// TIA Portal V17 export
// export: Created 2022-12-09T10:51:17.8914312Z, ExportSetting WithDefaults, DisplayName Totally Integrated Automation Portal, DisplayVersion V17 Update 5, DisplayName TIA Portal Openness, DisplayVersion V17 Update 5, DisplayName TIA Portal Version Control Interface, DisplayVersion V17, DisplayName Simotion SCOUT TIA, DisplayVersion 5.4.3.0, DisplayName SINAMICS Startdrive Advanced, DisplayVersion V17 SP1, DisplayName SINAMICS Startdrive G130, G150, S120, S150, SINAMICS MV, S210, DisplayVersion V17 SP1, DisplayName SINAMICS Startdrive G110M, G120, G120C, G120D, G120P, G115D, DisplayVersion V17 SP1, DisplayName STEP 7 Professional, DisplayVersion V17 Update 5, DisplayName STEP 7 Safety, DisplayVersion V17, DisplayName WinCC Advanced, DisplayVersion V17 Update 5
TYPE "UDT_OMAC_GlobalData"
// stored: IsFailsafeCompliant false
   STRUCT
      FirstCycle { ExternalAccessible := 'False'; ExternalVisible := 'False'; ExternalWritable := 'False'} : Bool := true;
      UnitMode : DInt;   // requested unit mode
      UnitModeChangeRequest : Bool := false;
      CntrlCmd : DInt;   // requested state
      CmdChangeRequest : Bool := false;   // request change in state
      enableBooleanInterface : Bool := false;
      ProductionModeRequest : Bool := false;
      MaintenanceModeRequest : Bool := false;
      ManualModeRequest : Bool := false;
      ChangeOverModeRequest : Bool := false;
      CleanModeRequest : Bool := false;
      SetUpModeRequest : Bool := false;
      EmptyOutModeRequest : Bool := false;
      OEMSpecificModeRequest : Bool := false;
      UserMode01Request : Bool := false;
      UserMode02Request : Bool := false;
      UserMode03Request : Bool := false;
      UserMode04Request : Bool := false;
      UserMode05Request : Bool := false;
      ResetCmdRequest : Bool := false;
      StartCmdRequest : Bool := false;
      StopCmdRequest : Bool := false;
      HoldCmdRequest : Bool := false;
      UnholdCmdRequest : Bool := false;
      SuspendCmdRequest : Bool := false;
      UnsuspendCmdRequest : Bool := false;
      AbortCmdRequest : Bool := false;
      ClearCmdRequest : Bool := false;
      CompleteCmdRequest : Bool := false;
      SC : Struct
         UNDEFINED : Bool;
         CLEARING : Bool;
         STOPPED : Bool;
         STARTING : Bool;
         IDLE : Bool;
         SUSPENDED : Bool;
         EXECUTE : Bool;
         STOPPING : Bool;
         ABORTING : Bool;
         ABORTED : Bool;
         HOLDING : Bool;
         HELD : Bool;
         UNHOLDING : Bool;
         SUSPENDING : Bool;
         UNSUSPENDING : Bool;
         RESETTING : Bool;
         COMPLETING : Bool;
         COMPLETE : Bool;
      END_STRUCT;
      configuration { S7_SetPoint := 'True'} : "UDT_OMAC_Configuration";
      UnitModeCurrent : DInt := 0;   // current mode
      UnitModeRequested : DInt := 0;   // requested unit mode
      UnitModeChangeInProcess : Bool := false;   // unit mode change in process
      StateCurrent : DInt := 0;   // current state
      StateRequested : DInt := 0;   // requested state
      StateChangeInProcess : Bool := false;   // state change in process
      ProductionModeActive : Bool := false;
      MaintenanceModeActive : Bool := false;
      ManualModeActive : Bool := false;
      ChangeOverModeActive : Bool := false;
      CleanModeRequestActive : Bool := false;
      SetUpModeRequestActive : Bool := false;
      EmptyOutModeRequestActive : Bool := false;
      OEMSpecificModeRequestActive : Bool := false;
      SpareModeActive : Bool;
      UserMode01Active : Bool := false;
      UserMode02Active : Bool := false;
      UserMode03Active : Bool := false;
      UserMode04Active : Bool := false;
      UserMode05Active : Bool := false;
      ClearingStateActive : Bool := false;
      StoppedStateActive : Bool := false;
      StartingStateActive : Bool := false;
      IdleStateActive : Bool := false;
      SuspendedStateActive : Bool := false;
      ExecuteStateActive : Bool := false;
      StoppingStateActive : Bool := false;
      AbortingStateActive : Bool := false;
      AbortedStateActive : Bool := false;
      HoldingStateActive : Bool := false;
      HeldStateActive : Bool := false;
      UnholdingStateActive : Bool := false;
      SuspendingStateActive : Bool := false;
      UnsuspendingStateActive : Bool := false;
      ResettingStateActive : Bool := false;
      CompletingStateActive : Bool := false;
      CompleteStateActive : Bool := false;
      StatesDisabled : DInt;
      diagnostics { S7_SetPoint := 'True'} : "UDT_OMAC_Diagnostics";
      diagnosticsBufferIndexForHMI : Int;
      diagnosticsBufferEntryForHMI { S7_SetPoint := 'True'} : "UDT_OMAC_DiagnosticsEntry";
      namesConfiguration { S7_SetPoint := 'True'} : "UDT_OMAC_NamesConfiguration";
      language : Int;
      unitModeCurrentName : String[18];
      stateCurrentName : String[16];
   END_STRUCT;
END_TYPE
